TEXTLIST languageSupport
  axesAvailable = 'PLC Axes available: %d' | Test: 'Alt language'
  velocity = 'Velocity:'
  actposition = 'Actual Position:'
  enable = 'Enable Axis'
  enFW = 'Fwd Enable'
  enBW = 'Bwd Enable'
  axisSel = 'Axis Selected:'
  actVelocity = 'Actual Velocity:'
  errID = 'Error ID:'
  bEnabled = 'Axis Enabled'
  bCommandAborted = 'Command Aborted'
  bBusy = 'Busy'
  bDone = 'Command Done'
  bResetDone = 'Reset Complete'
  bHomed = 'Calibrated'
  bFwEnabled = 'Fwd movement enabled'
  bBwEnabled = 'Bwd movement enabled'
  bError = 'Error'
  fVelocity = 'Target Velocity:'
  fAcceleration = 'Target Accel.:'
  fDeceleration = 'Target Decel.:'
  fPosition = 'Target Position:'
  moveAbsolute = 'Absolute position move'
  toggle = 'Toggle'
  moveVelocity = 'Constant velocity move'
  bExecute = 'Motion function executed'
  moveRelative = 'Relative position move'
  moveModulo = 'Modulo position move'
  reset = 'Reset axis'
  stop = 'Stop motion'
  jogBw = 'Jog Backward'
  jogFw = 'Jog Forward'
  bGeared = 'In Gear'
  masterGear = 'Master Axis'
  gearRatio = 'Gear Ratio'
  gearIn = 'Gear In'
  gearOut = 'Gear Out'
  eHomeToLimit_Bwd = 'Bwd Limit'
  eHomeToLimit_Fwd = 'Fwd Limit'
  eHomeToRef_Bwd = 'Home Switch Bwd '
  eHomeToRef_Fwd = 'Home Switch Fwd '
  eHomeToEncPulse_Bwd = 'Enc Index Bwd '
  eHomeToEncPulse_Fwd = 'Enc Index Fwd'
  eHomeToEncPulse_viaBwdLimit = 'Enc Index via Bwd Limit'
  eHomeToEncPulse_viaFwdLimit = 'Enc Index via Fwd Limit'
  eHomeToBlock_Bwd = 'Home To Block Bwd'
  eHomeToBlock_Fwd = 'Home To Block Fwd'
  eHomeDirect = 'Home Direct'
  fHomePosition = 'Set Pos after Homing'
  fHomeFinishDistance = 'Move after Homing'
  halt = 'Halt Motion'
  bInterlockBwd = 'Interlock Bwd'
  bInterlockFwd = 'Interlock Fwd'
  Home = 'HOME'
  eWriteParameter = 'Write Parameter'
  eReadParameter = 'Read Parameter'
  fWriteAxisParameter = 'Parameter to write'
  fReadAxisParameter = 'Parameter'
  bLocalMode = 'Local Mode'
  bInVelocity = 'Target velocity reached'
  bHighTempAxisDisabled = 'Disabled by High Temp '
  fActualTemp = 'Actual Temp'
  bHWMaskActive = 'HW Mask Active'
  bMoving = 'Moving'
  bEnableStopWithAnyLimitSwitch = 'Stop at any Limit Switch'
  eWriteCoEParameter = 'Write CoE Parameter'
  eReadCoEParameter = 'Read CoE Parameter'
  fWriteCoEParameter = 'CoE param. to write'
  fReadCoEParameter = 'CoE Parameter'
  enSoftLimBw = 'Soft Lim Bwd On'
  enSoftLimFw = 'Soft Lim Fwd On'
  disSoftLimBw = 'Soft Lim Bwd Off'
  disSoftLimFw = 'Soft Lim Fwd Off'
  SWLimitSwitches = 'SW Limit Switches'
  CommandHandler = 'Command Handler'
  bCommandHandlerBufferingCommand = 'Buffering Command'
  bAxisReadyToMove = 'Axis Ready To Move'
  bCommandHandlerTimeoutError = 'Timeout Cmd Handler'
  tCommandHandlerTimeout = 'Timeout Buffering Command'
  bCommandHandlerMovePermit = 'Move Permit'
  Airpad = 'Airpad'
  bAirpadConnected = 'Airpad Connected'
  bAirpadFeedbackConnected = 'Feedback Connected'
  bAirpadManualControl = 'Allow Manual Control'
  bAirpadManualPressureOn = 'Pressure On / Off'
  tAirpadOnDelayTime = 'Airpad On Delay'
  bAirpadReady = 'Airpad Ready'
  bAirpadPressurized = 'Feedback: Pressurized'
  bAirpadPressureError = 'Pressure Error'
  bAirpadTimeoutError = 'Pressurize Timeout'
  tAirpadPressurizeTimeout = 'Timeout Pressurizing Airpad'
  tAirpadDepressurizeTimeout = 'Timeout Depressurizing Airpad'
  ExternalBrake = 'External Brake'
  bExternalBrakeConnected = 'External Brake Connected'
  bExternalBrakeFeedbackConnected = 'Feedback Connected'
  tBrakeOpenDelayTime = 'Brake Release Delay'
  tBrakeCloseAheadTime = 'Amplifier Off Delay'
  tBrakeOpeningTimeoutWhenFeedback = 'Opening Timeout When Feedback'
  bExternalBrakeReady = 'External Brake Ready'
  bBrakeReleased = 'Feedback: Released'
  bExternalBrakeFailure = 'Brake Error'
  bExternalBrakeTimeoutError = 'Timeout Releasing Brake'
  nSoEDiagID = 'SoE Drive Diagnostic ID'
  nSoEErrorID = 'SoE Drive Error ID'
  bSoEDriveDeviceError = 'DriveDeviceError'
  fMinSoftLimit = 'Current Soft Limit Min '
  fMaxSoftLimit = 'Current Soft Limit Max'
  fWriteSoftLimitMin = 'Set Soft Limit Min'
  fWriteSoftLimitMax = 'Set Soft Limit Max'
  bCommandHandlerReleasedCommand = 'Move Command Released'
   = ''
END_TEXTLIST

(* stored: Version 1.1.0.1
   TextList languageSupport: Id {5d3fdc2f-5bea-44d3-8108-bdef8127e821} *)
